(* PLC project Sin nombre, Desconocido Sin nombre 1 *)
(* stored: creationDateTime 2022-10-17T16:56:25, modificationDateTime 2025-10-24T16:01:41 *)

PROGRAM program0
  VAR
    Led AT %QX0.0 : BOOL := 0;
    Sensor AT %IX0.1 : BOOL := 0;
  END_VAR
  VAR
    TP0 : TP;
    TOF0 : TOF;
    TP1 : TP;
  END_VAR

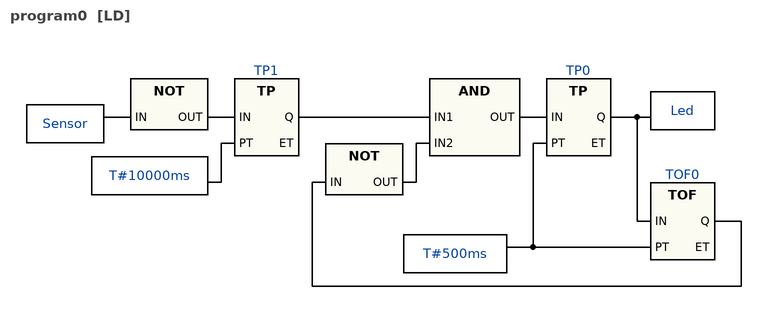
(* LD diagram, written out as Structured Text *)
TP1(IN := NOT Sensor, PT := T#10000ms);
TOF0(IN := TP0.Q, PT := T#500ms);
TP0(IN := TP1.Q AND NOT TOF0.Q, PT := T#500ms);
Led := TP0.Q;
END_PROGRAM

CONFIGURATION Config0
  RESOURCE Res0 ON PLC
    TASK task0(INTERVAL := T#20ms, PRIORITY := 0);
    PROGRAM instance0 WITH task0 : program0;
  END_RESOURCE
END_CONFIGURATION
